(* PLC project Adressering.ecp, WAGO e!COCKPIT e!COCKPIT *)
(* stored: creationDateTime 2021-01-18T14:20:23.2110188, modificationDateTime 2021-01-18T11:51:27.6823754 *)

TYPE dtRomtype_11111111 : STRUCT
  RB601_V : BOOL;  (* Bevegelse *)
  RB601_HVAC : BOOL;  (* HVAC signal *)
  RT601_CT : REAL;  (* Rom temperatur *)
  RT601_SP_D : REAL;  (* Temperatur SP *)
  RT601_SP_S : REAL;  (* Temperatur SP standby *)
  RT601_SP_N : REAL;  (* Temperatur SP nattsenk *)
  RT601_SP_F : REAL;  (* Temperatur SP frostsikring *)
  RT601_CS : REAL;  (* Aktivt temperatur SP *)
  OPM : INT;  (* Rom modus *)
  OPM_CV : INT;  (* Rom modus verdi *)
  RY601_CV : REAL;  (* Co2 Nivaa *)
  RY601_SP : REAL;  (* Co2 SP *)
  RY601_OP : REAL;  (* Co2 paadrag *)
  LH601_OP : REAL;  (* Varmepaadrag *)
  LH601_MAN : BOOL;  (* Force LH *)
  LH601_CMD : BOOL;  (* LH601_CMD *)
  LC601_OP : REAL;  (* LC601_OP *)
  LC601_SP : REAL;  (* LC SP *)
  LC601_MAN : BOOL;  (* Force LC *)
  LC601_CMD : BOOL;  (* LC601_CMD *)
END_STRUCT;
END_TYPE

{attribute 'qualified_only'}
VAR_GLOBAL  (* STLV59_563 *)
  STLV59_A_563_RB001_HVAC : BOOL;  (* HVAC signal for PLS *)
  STLV59_A_563_KNX_Card_1_Status : BOOL;  (* KNX kort 1 status *)
  STLV59_A_563_001 : dtRomtype_11111111;  (* Placeholder_1æøå *)
END_VAR

FUNCTION_BLOCK fbRomtype_11111111
  VAR_INPUT
    RB601_HVAC : BOOL;
    RT601_CT : REAL;
    RT601_SP_D : REAL;
    RT601_SP_S : REAL;
    RT601_SP_N : REAL;
    RT601_SP_F : REAL;
    OPM : INT;
    RY601_CV : REAL;
    RY601_SP : REAL;
    LH601_MAN : BOOL;
    LC601_SP : REAL;
    LC601_MAN : BOOL;
  END_VAR
  VAR_OUTPUT
    OPM_CV : INT;
    RT601_CS : REAL;
    RY601_OP : REAL;
    LH601_OP : REAL;
    LH601_CMD : BOOL;
    LC601_OP : REAL;
    LC601_CMD : BOOL;
  END_VAR

(* CFC diagram, written out as Structured Text *)
END_FUNCTION_BLOCK

FUNCTION_BLOCK fbSE_Hyst
  VAR_INPUT
    rIn : REAL;
    rOn : REAL;
    rOff : REAL;
  END_VAR
  VAR_OUTPUT
    xOut : BOOL;
  END_VAR

					xOut:= ((rOn > rOff AND (rIn >= rOn OR (xOut AND rIn > rOff)))	OR		(rOn <rOff AND (rIn <= rOn OR (xOut AND rIn <rOff))));
				
END_FUNCTION_BLOCK

PROGRAM PRG_KNX_563_1
  VAR
    i : INT := 0;  (* Felles *)
    Interval : TON := (PT := TIME#2m0s0ms);
    typDPT : typDPT;
    KNX_master_1 : WagoAppKNX.FbKNX_Master;  (* Master *)
    M1_001_001_RB601_V : fbDPT_Switch_pro;  (* 001 *)
    M1_002_001_RB601_HVAC : fbDPT_Switch_pro;
    M1_003_001_RT601_CT : fbDPT_Value_Temp_pro;
    M1_004_001_RY601_CV : fbDPT_Value_AirQuality_pro;
    M1_005_001_LH601_OP : fbDPT_Scaling_pro;
    M1_006_001_LH601_CMD : fbDPT_Switch_pro;
    M1_007_001_LC601_OP : fbDPT_Scaling_pro;
    M1_008_001_LC601_CMD : fbDPT_Switch_pro;
  END_VAR
  VAR  (* added by the conversion: wires and edge detectors of the diagram *)
    _ADD9_OUT : INT;
    _GT15_OUT : BOOL;
    _MOVE19_ENO : BOOL;
    _MOVE19_OUT : INT;
    _MOVE46_ENO : BOOL;
    _MOVE46_OUT : ANY;
    _MOVE59_ENO : BOOL;
    _MOVE59_OUT : ANY;
    _MOVE72_ENO : BOOL;
    _MOVE72_OUT : ANY;
    _MOVE85_ENO : BOOL;
    _MOVE85_OUT : ANY;
  END_VAR

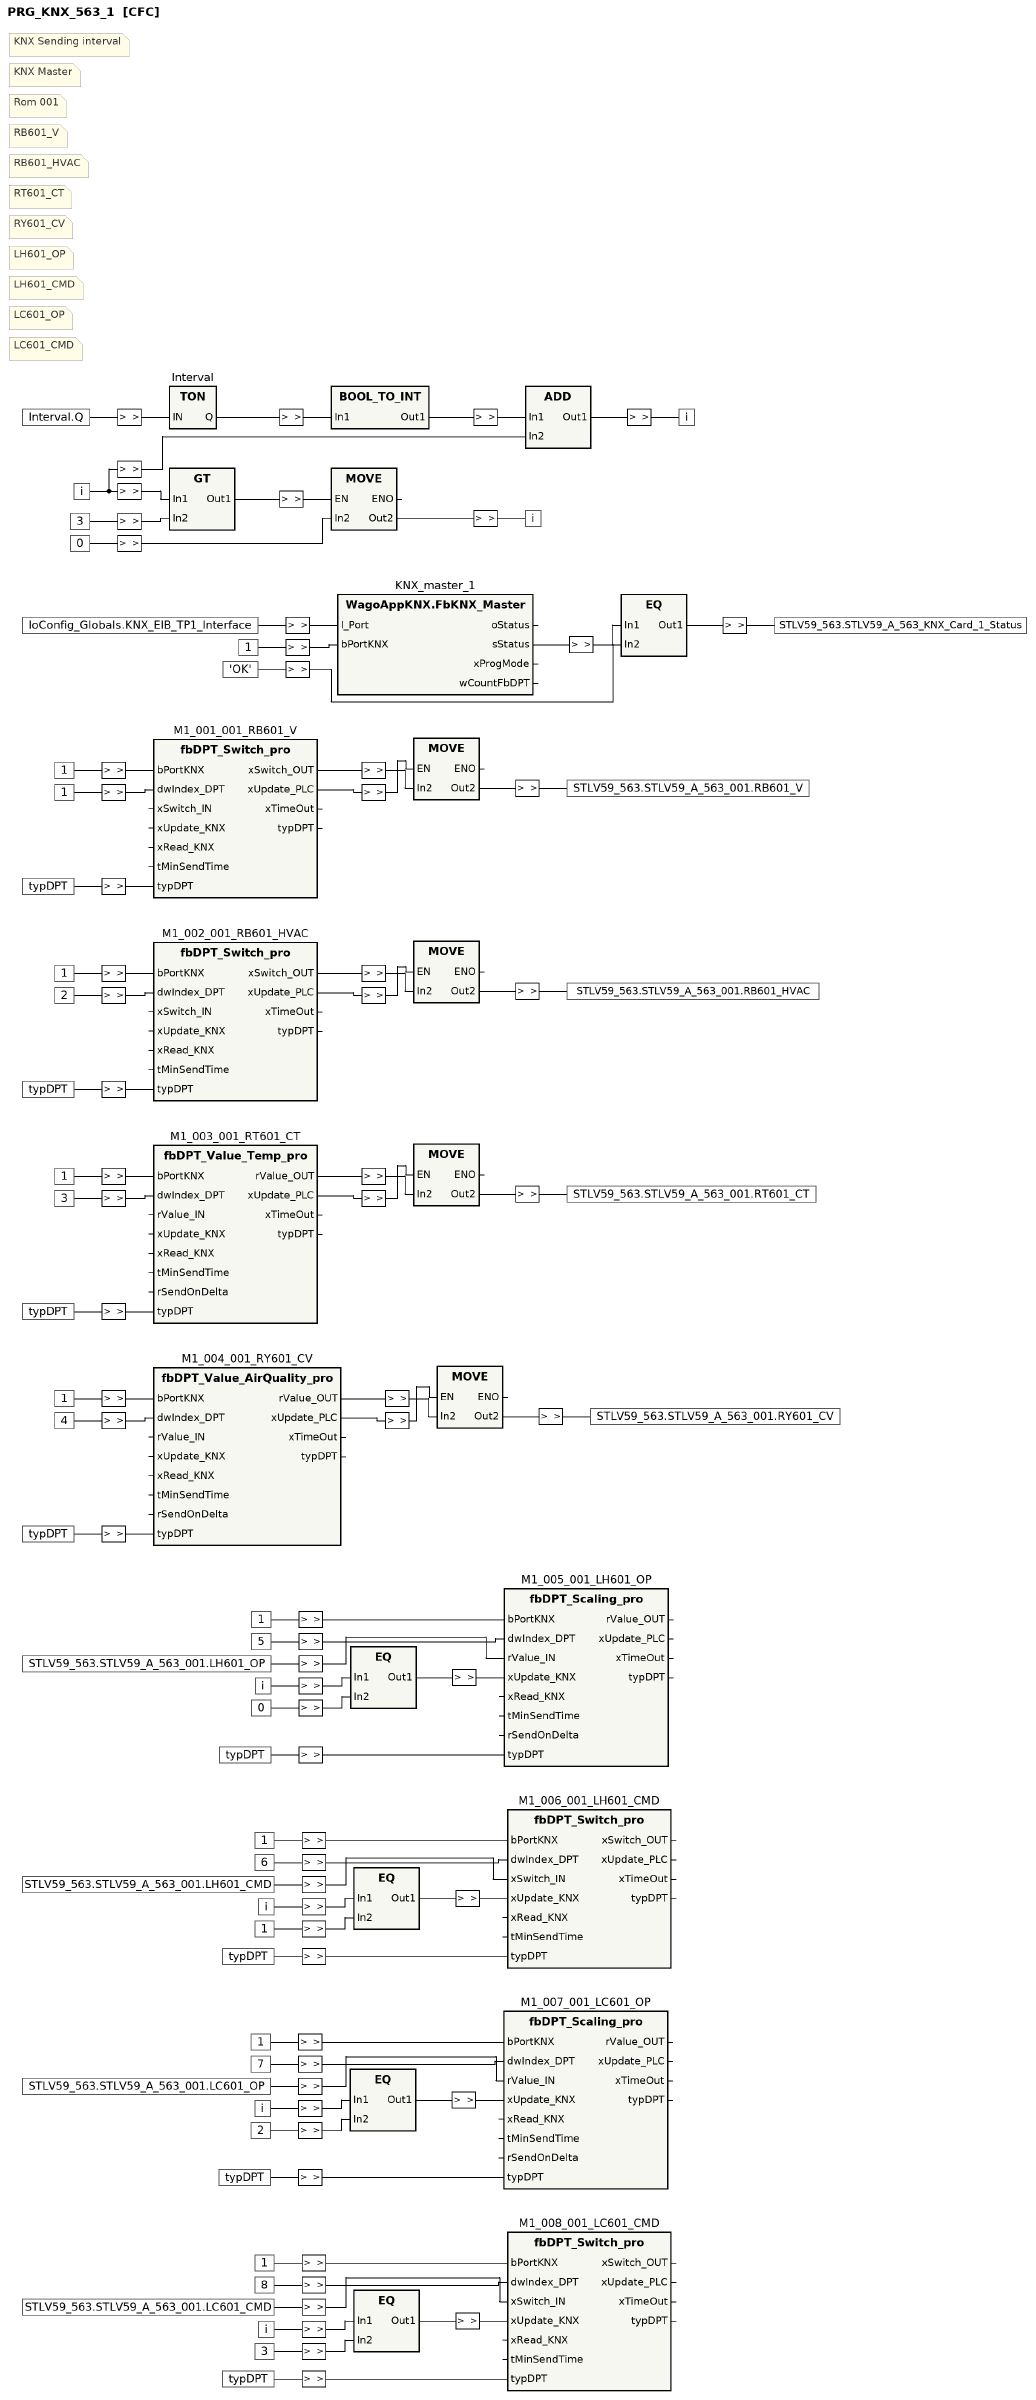
(* CFC diagram, written out as Structured Text *)
(* KNX Sending interval *)
(* KNX Master *)
Interval(IN := Interval.Q);
_ADD9_OUT := BOOL_TO_INT(Interval.Q) + i;
i := _ADD9_OUT;
_GT15_OUT := i > 3;
_MOVE19_OUT := MOVE(EN := _GT15_OUT, IN := 0, ENO => _MOVE19_ENO);
IF _MOVE19_ENO THEN i := _MOVE19_OUT; END_IF;
KNX_master_1(I_Port := IoConfig_Globals.KNX_EIB_TP1_Interface, bPortKNX := 1);
STLV59_563.STLV59_A_563_KNX_Card_1_Status := KNX_master_1.sStatus = 'OK';
(* Rom 001 *)
(* RB601_V *)
(* RB601_HVAC *)
M1_001_001_RB601_V(bPortKNX := 1, dwIndex_DPT := 1, typDPT := typDPT);
_MOVE46_OUT := MOVE(EN := M1_001_001_RB601_V.xUpdate_PLC, IN := M1_001_001_RB601_V.xSwitch_OUT, ENO => _MOVE46_ENO);
IF _MOVE46_ENO THEN STLV59_563.STLV59_A_563_001.RB601_V := _MOVE46_OUT; END_IF;
M1_002_001_RB601_HVAC(bPortKNX := 1, dwIndex_DPT := 2, typDPT := typDPT);
_MOVE59_OUT := MOVE(EN := M1_002_001_RB601_HVAC.xUpdate_PLC, IN := M1_002_001_RB601_HVAC.xSwitch_OUT, ENO => _MOVE59_ENO);
IF _MOVE59_ENO THEN STLV59_563.STLV59_A_563_001.RB601_HVAC := _MOVE59_OUT; END_IF;
(* RT601_CT *)
(* RY601_CV *)
M1_003_001_RT601_CT(bPortKNX := 1, dwIndex_DPT := 3, typDPT := typDPT);
_MOVE72_OUT := MOVE(EN := M1_003_001_RT601_CT.xUpdate_PLC, IN := M1_003_001_RT601_CT.rValue_OUT, ENO => _MOVE72_ENO);
IF _MOVE72_ENO THEN STLV59_563.STLV59_A_563_001.RT601_CT := _MOVE72_OUT; END_IF;
M1_004_001_RY601_CV(bPortKNX := 1, dwIndex_DPT := 4, typDPT := typDPT);
_MOVE85_OUT := MOVE(EN := M1_004_001_RY601_CV.xUpdate_PLC, IN := M1_004_001_RY601_CV.rValue_OUT, ENO => _MOVE85_ENO);
IF _MOVE85_ENO THEN STLV59_563.STLV59_A_563_001.RY601_CV := _MOVE85_OUT; END_IF;
(* LH601_OP *)
(* LH601_CMD *)
M1_005_001_LH601_OP(bPortKNX := 1, dwIndex_DPT := 5, rValue_IN := STLV59_563.STLV59_A_563_001.LH601_OP, xUpdate_KNX := i = 0, typDPT := typDPT);
M1_006_001_LH601_CMD(bPortKNX := 1, dwIndex_DPT := 6, xSwitch_IN := STLV59_563.STLV59_A_563_001.LH601_CMD, xUpdate_KNX := i = 1, typDPT := typDPT);
(* LC601_OP *)
(* LC601_CMD *)
M1_007_001_LC601_OP(bPortKNX := 1, dwIndex_DPT := 7, rValue_IN := STLV59_563.STLV59_A_563_001.LC601_OP, xUpdate_KNX := i = 2, typDPT := typDPT);
M1_008_001_LC601_CMD(bPortKNX := 1, dwIndex_DPT := 8, xSwitch_IN := STLV59_563.STLV59_A_563_001.LC601_CMD, xUpdate_KNX := i = 3, typDPT := typDPT);
END_PROGRAM

PROGRAM PRG_563_Romstyring
  VAR
    Rom_001 : fbRomtype_11111111;  (* 001 *)
  END_VAR

(* CFC diagram, written out as Structured Text *)
(* Rom 001 *)
Rom_001(RB601_HVAC := STLV59_563.STLV59_A_563_001.RB601_HVAC, RT601_CT := STLV59_563.STLV59_A_563_001.RT601_CT, RT601_SP_D := STLV59_563.STLV59_A_563_001.RT601_SP_D, RT601_SP_S := STLV59_563.STLV59_A_563_001.RT601_SP_S, RT601_SP_N := STLV59_563.STLV59_A_563_001.RT601_SP_N, RT601_SP_F := STLV59_563.STLV59_A_563_001.RT601_SP_F, OPM := STLV59_563.STLV59_A_563_001.OPM, RY601_CV := STLV59_563.STLV59_A_563_001.RY601_CV, RY601_SP := STLV59_563.STLV59_A_563_001.RY601_SP, LH601_MAN := STLV59_563.STLV59_A_563_001.LH601_MAN, LC601_SP := STLV59_563.STLV59_A_563_001.LC601_SP, LC601_MAN := STLV59_563.STLV59_A_563_001.LC601_MAN);
STLV59_563.STLV59_A_563_001.OPM_CV := Rom_001.OPM_CV;
STLV59_563.STLV59_A_563_001.RT601_CS := Rom_001.RT601_CS;
STLV59_563.STLV59_A_563_001.RY601_OP := Rom_001.RY601_OP;
STLV59_563.STLV59_A_563_001.LH601_OP := Rom_001.LH601_OP;
STLV59_563.STLV59_A_563_001.LH601_CMD := Rom_001.LH601_CMD;
STLV59_563.STLV59_A_563_001.LC601_OP := Rom_001.LC601_OP;
STLV59_563.STLV59_A_563_001.LC601_CMD := Rom_001.LC601_CMD;
END_PROGRAM

PROGRAM PRG_360_HVAC

	STLV59_563.STLV59_A_563_RB001_HVAC:=
(
	STLV59_563.STLV59_A_563_001.RB601_HVAC
);
END_PROGRAM
